{attribute 'qualified_only'}
{attribute 'strict'}
{attribute 'to_string'}
TYPE E_RequestMode :
(
	{attribute 'hide'}
    Undefined   := 0,
	Automatic   := 1,
    Semiauto    := 2,
	Manual		:= 3
);
END_TYPE

(* stored: Version 1.1.0.1
   DUT E_RequestMode: Id {45515ad4-f759-0ed7-2dc8-c62d4b040a65} *)
